PROGRAM MAIN
VAR
		
	sSrvNetID		: T_AmsNetID	:= '';
	bScannerEnable	: BOOL 			:= FALSE;
//	bLaserEnable	: BOOL 			:= TRUE;
	bLog			: BOOL			:= FALSE;
	fbClient_ABC 	: FB_Client 	:= ( sRemoteHost := '192.168.1.177',
										 nRemotePort := 8500,
										 sPrefix := '' );
										
	fbCloseAll		: FB_SocketCloseAll;
	bInitialize		: BOOL := TRUE;
	bConnected		: BOOL;
	nErrId			: UDINT;
	data_send_flag  : BOOL;
	Msg			: STRING := '';
	Send_msg		: STRING := '';
	Received_msg	: STRING := '';

END_VAR

	fbCloseAll( sSrvNetID := sSrvNetID, bExecute:= bInitialize );
	IF fbCloseAll.bBusy OR fbCloseAll.bError THEN
		nErrId := fbCloseAll.nErrId;
		RETURN;
	END_IF
	
	bInitialize := FALSE;
	fbClient_ABC	( sSrvNetId := sSrvNetID, bEnable := bScannerEnable	, bLog := bLog, bConnected => bConnected );
	
	IF data_send_flag THEN
		Send_msg := CONCAT(Msg, '$R');
		fbClient_ABC.fbTx.AddTail( sPut := Send_msg); //$R = Carriage Return [CR]
		data_send_flag := false;
	END_IF
	
	Received_msg := fbClient_ABC.RxText;

END_PROGRAM

(* stored: Version 1.1.0.1, ProductVersion 3.1.4024.12
   POU MAIN: Id {34528779-84b6-44e4-a437-083f290810e9}, SpecialFunc None *)
